// SIMATIC S7-200 project (STEP 7-Micro/WIN), CPU 221 REL 01.10

SYMBOL_TABLE USER1
e10              M0.0
e11              M0.1
e12              M0.2
e13              M0.3
e14              M0.4
e15              M0.5
e20              M1.0
e21              M1.1
e22              M1.2
e23              M1.3
e24              M1.4
e25              M1.5
e26              M1.6
e27              M1.7
e28              M2.0
PG               Q1.0
PM               Q1.1
PP               Q1.2
S1               I0.0
S2               I0.1
S3               I0.2
S4               I0.3
S5               I0.4
S6               I0.5
S7               I0.6
S8               I1.7
M1               Q0.0
M2               Q0.1
V1               Q0.2
V2               Q0.3
V3               Q0.4
BPG              I1.2
BPM              I1.3
BPP              I1.4
BRC              I1.5
ev1              I1.0
ev2              I1.1
ev3              I1.6
CG               M2.1
CM               M2.2
END_SYMBOL_TABLE

ORGANIZATION_BLOCK MAIN:OB1
TITLE=PROGRAM COMMENTS
BEGIN
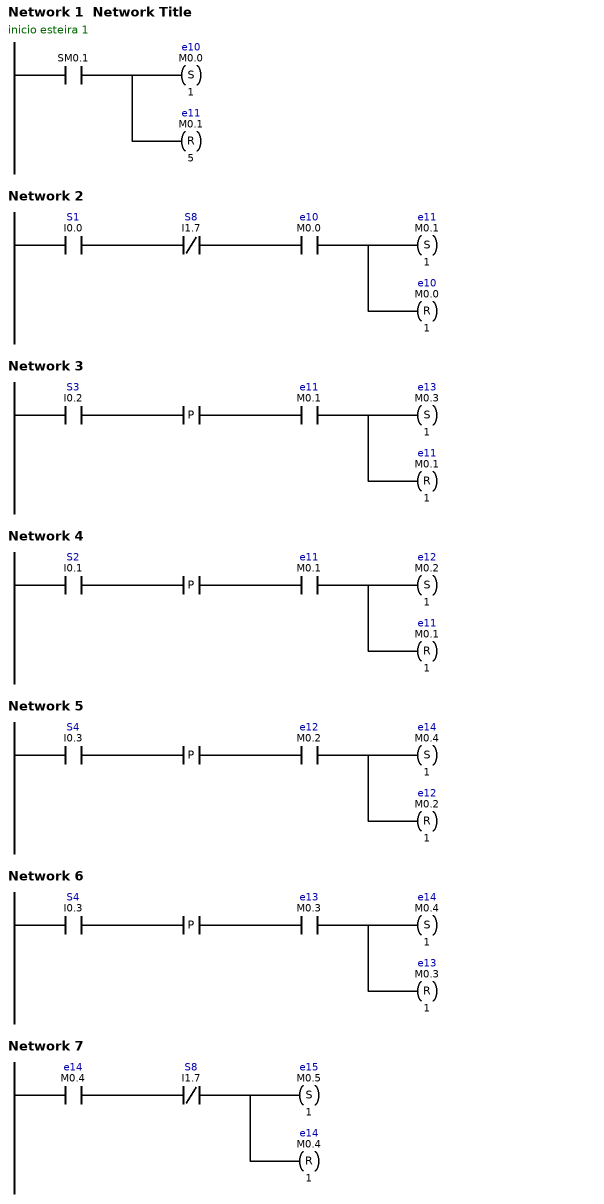
Network 1 // Network Title
// inicio esteira 1
LD     SM0.1
S      e10:M0.0, 1
R      e11:M0.1, 5
Network 2
LD     S1:I0.0
AN     S8:I1.7
A      e10:M0.0
S      e11:M0.1, 1
R      e10:M0.0, 1
Network 3
LD     S3:I0.2
EU
A      e11:M0.1
S      e13:M0.3, 1
R      e11:M0.1, 1
Network 4
LD     S2:I0.1
EU
A      e11:M0.1
S      e12:M0.2, 1
R      e11:M0.1, 1
Network 5
LD     S4:I0.3
EU
A      e12:M0.2
S      e14:M0.4, 1
R      e12:M0.2, 1
Network 6
LD     S4:I0.3
EU
A      e13:M0.3
S      e14:M0.4, 1
R      e13:M0.3, 1
Network 7
LD     e14:M0.4
AN     S8:I1.7
S      e15:M0.5, 1
R      e14:M0.4, 1
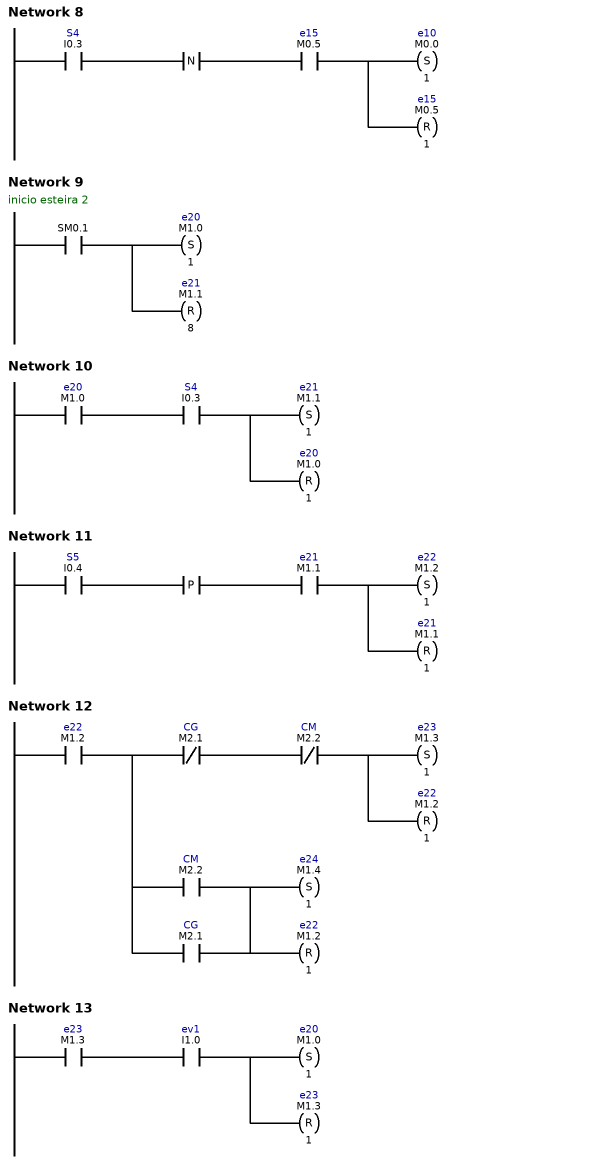
Network 8
LD     S4:I0.3
ED
A      e15:M0.5
S      e10:M0.0, 1
R      e15:M0.5, 1
Network 9
// inicio esteira 2
LD     SM0.1
S      e20:M1.0, 1
R      e21:M1.1, 8
Network 10
LD     e20:M1.0
A      S4:I0.3
S      e21:M1.1, 1
R      e20:M1.0, 1
Network 11
LD     S5:I0.4
EU
A      e21:M1.1
S      e22:M1.2, 1
R      e21:M1.1, 1
Network 12
LD     e22:M1.2
LPS
AN     CG:M2.1
AN     CM:M2.2
S      e23:M1.3, 1
R      e22:M1.2, 1
LPP
LD     CM:M2.2
O      CG:M2.1
ALD
S      e24:M1.4, 1
R      e22:M1.2, 1
Network 13
LD     e23:M1.3
A      ev1:I1.0
S      e20:M1.0, 1
R      e23:M1.3, 1
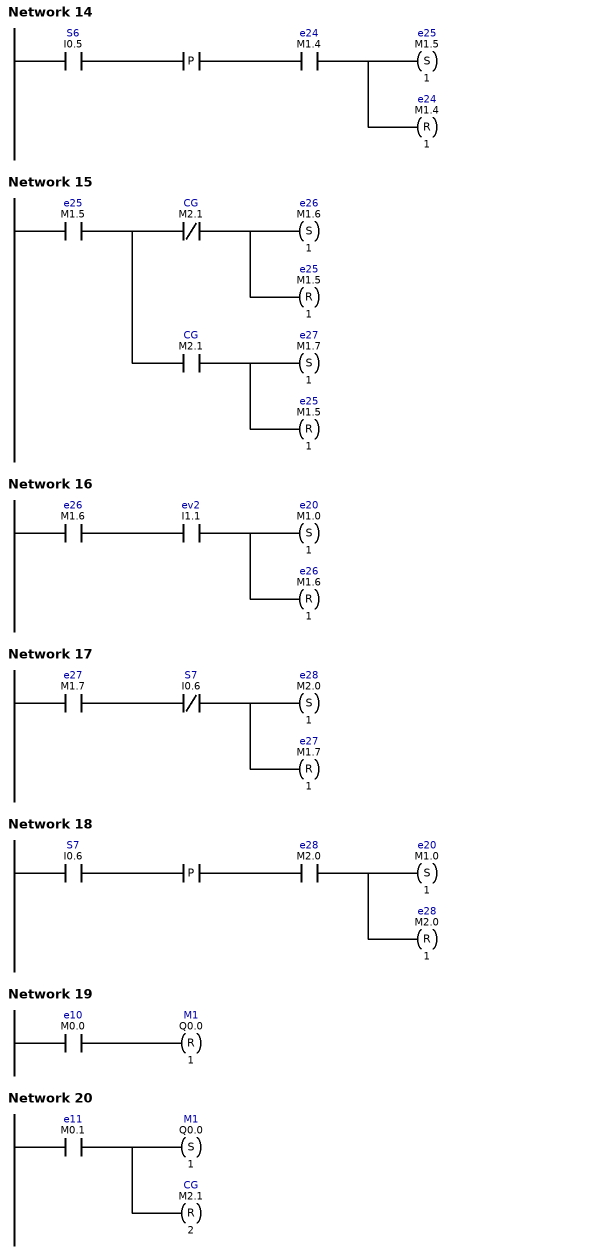
Network 14
LD     S6:I0.5
EU
A      e24:M1.4
S      e25:M1.5, 1
R      e24:M1.4, 1
Network 15
LD     e25:M1.5
LPS
AN     CG:M2.1
S      e26:M1.6, 1
R      e25:M1.5, 1
LPP
A      CG:M2.1
S      e27:M1.7, 1
R      e25:M1.5, 1
Network 16
LD     e26:M1.6
A      ev2:I1.1
S      e20:M1.0, 1
R      e26:M1.6, 1
Network 17
LD     e27:M1.7
AN     S7:I0.6
S      e28:M2.0, 1
R      e27:M1.7, 1
Network 18
LD     S7:I0.6
EU
A      e28:M2.0
S      e20:M1.0, 1
R      e28:M2.0, 1
Network 19
LD     e10:M0.0
R      M1:Q0.0, 1
Network 20
LD     e11:M0.1
S      M1:Q0.0, 1
R      CG:M2.1, 2
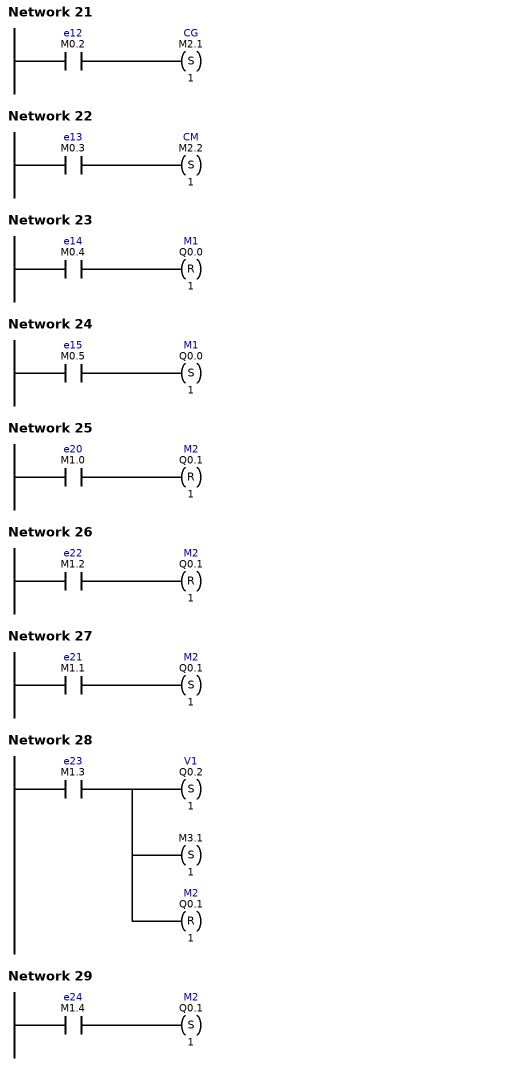
Network 21
LD     e12:M0.2
S      CG:M2.1, 1
Network 22
LD     e13:M0.3
S      CM:M2.2, 1
Network 23
LD     e14:M0.4
R      M1:Q0.0, 1
Network 24
LD     e15:M0.5
S      M1:Q0.0, 1
Network 25
LD     e20:M1.0
R      M2:Q0.1, 1
Network 26
LD     e22:M1.2
R      M2:Q0.1, 1
Network 27
LD     e21:M1.1
S      M2:Q0.1, 1
Network 28
LD     e23:M1.3
S      V1:Q0.2, 1
S      M3.1, 1
R      M2:Q0.1, 1
Network 29
LD     e24:M1.4
S      M2:Q0.1, 1
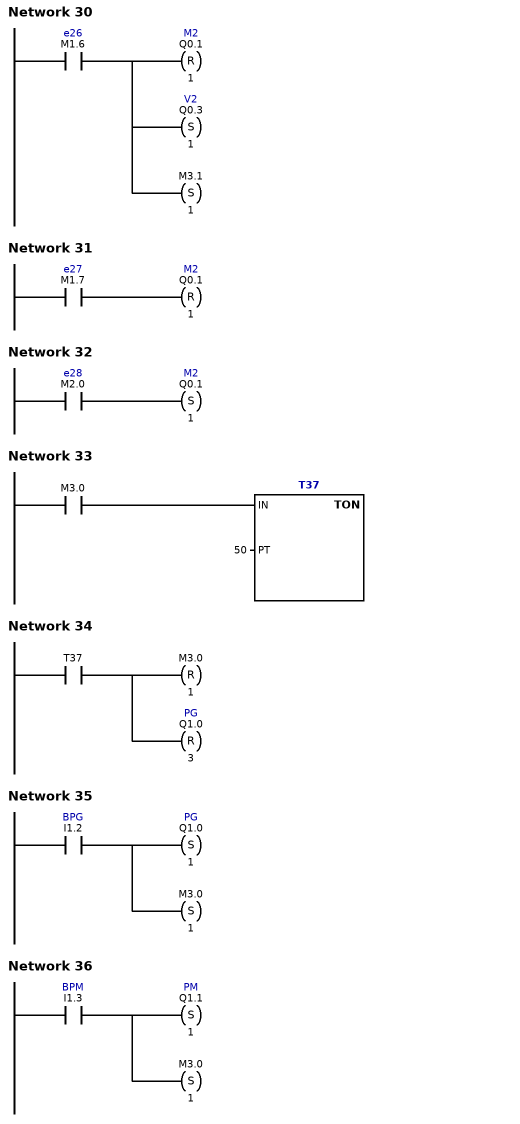
Network 30
LD     e26:M1.6
R      M2:Q0.1, 1
S      V2:Q0.3, 1
S      M3.1, 1
Network 31
LD     e27:M1.7
R      M2:Q0.1, 1
Network 32
LD     e28:M2.0
S      M2:Q0.1, 1
Network 33
LD     M3.0
TON    T37, 50
Network 34
LD     T37
R      M3.0, 1
R      PG:Q1.0, 3
Network 35
LD     BPG:I1.2
S      PG:Q1.0, 1
S      M3.0, 1
Network 36
LD     BPM:I1.3
S      PM:Q1.1, 1
S      M3.0, 1
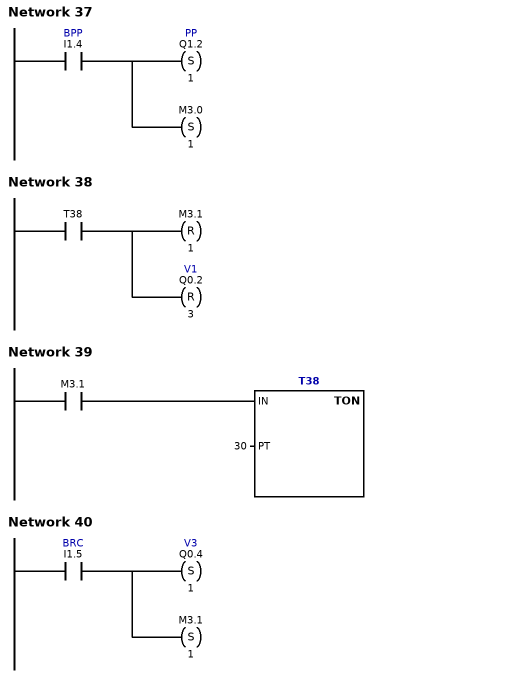
Network 37
LD     BPP:I1.4
S      PP:Q1.2, 1
S      M3.0, 1
Network 38
LD     T38
R      M3.1, 1
R      V1:Q0.2, 3
Network 39
LD     M3.1
TON    T38, 30
Network 40
LD     BRC:I1.5
S      V3:Q0.4, 1
S      M3.1, 1
END_ORGANIZATION_BLOCK
